Staubli VAL3: setListOfItems.pgx

public program setListOfItems(num x_nListNumber, string& x_sItemList[], num& x_nError[])
begin
  // This program fills a list object with items
  //
  // Input Param
  //  x_nListNumber  : list number to fill
  //  x_sItemList    : Items to push into the List object
  //
  // Output Param
  //  x_Error : Error code
  //          = 3    : Variable pw:sListItemX doesn't exist (from listFilling)
  //
  //--------------------------------------------------------------
  //
  x_nError=0
  call pw:listFilling(x_nListNumber,x_sItemList,x_nError)
  if x_nError==0
    if size(pw:nListSize)<x_nListNumber+1
      resize(pw:nListSize,1,x_nListNumber+1)
    endIf
    pw:nListSize[x_nListNumber]=size(x_sItemList)
  else
    // Prepare clear text error message
    call ut:addNumToString(sErrMsgList[x_nError],sErrorMessage,"*",x_nListNumber)
  endIf
end
